FUNCTION_BLOCK CSMA
  (* Standard: 61499-2 *)
  (* Version 0.1, 2015-00-24, Jin, Jin-PC *)
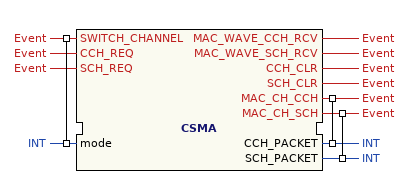
  EVENT_INPUT
    SWITCH_CHANNEL WITH mode;
    CCH_REQ;
    SCH_REQ;
  END_EVENT
  EVENT_OUTPUT
    MAC_WAVE_CCH_RCV;
    MAC_WAVE_SCH_RCV;
    CCH_CLR;
    SCH_CLR;
    MAC_CH_CCH WITH CCH_PACKET;
    MAC_CH_SCH WITH SCH_PACKET;
  END_EVENT
  VAR_INPUT
    mode : INT;
  END_VAR
  VAR_OUTPUT
    CCH_PACKET : INT;
    SCH_PACKET : INT;
  END_VAR
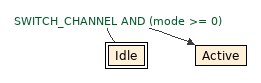
  EC_STATES
    Idle;
    Active;
  END_STATES
  EC_TRANSITIONS
    Idle TO Active := SWITCH_CHANNEL AND (mode >= 0);
  END_TRANSITIONS
END_FUNCTION_BLOCK
